// TIA Portal V19 export
DATA_BLOCK "PumpControl1"   // DB9
// stored: InstanceOfName Pump_Block, InstanceOfType FB
"Pump_Block"
   // VAR_INPUT
   //    Mode_Selection : Bool;
   //    Start_Manual : Bool;
   //    Stop_Manual : Bool;
   //    Start_Auto : Bool;
   //    Stop_Auto : Bool;
   //    Level_High : Bool;
   //    Level_Low : Bool;
   //    Set_Time_Start : DInt;
   //    Overload : Bool;
   //    Reset_Fault : Bool;
   // END_VAR
   // VAR_OUTPUT
   //    Pump_Run : Bool;
   //    Fault : Bool;
   //    Running_Auto_Mode : Bool;
   // END_VAR
   // VAR
   //    Timer_Start : IEC_TIMER;
   //    Start_Auto_Activated : Bool;
   // END_VAR
BEGIN
END_DATA_BLOCK
